TYPE Log_p_h :
STRUCT
	xDruck :=	 REAL; // log (Bar}
	yEnthalpie := REAL; // log (J)
END_STRUCT
END_TYPE

(* stored: Version 1.1.0.1, ProductVersion 3.1.4018.5
   DUT Log_p_h: Id {2f225f72-14f3-436c-87e9-0046cbe108e8} *)
